(* IEC 61131-3 sources: AutomationLab/ConveyerObject, 5 files *)

(* ---- ConveyerType.st ---- *)
TYPE ConveyerType :
STRUCT
	SensorA : BOOL;
	ComRotateLent : BOOL;
END_STRUCT
END_TYPE

(* ---- DT_Conveyer.st ---- *)
TYPE DT_Conveyer:
STRUCT
	// Коробка на конце ленты (от оптического датчика)
	BoxOnEndPosition: BOOL;
	// Команда на вращение ленты
	ComRotateLent: BOOL;
END_STRUCT
END_TYPE

(* ---- Conveyer_Main.st ---- *)
// ============================================
// ФУНКЦИОНАЛЬНЫЙ БЛОК — конвейер
// ============================================
FUNCTION_BLOCK Conveyer_Main
VAR_INPUT
END_VAR

VAR_OUTPUT
END_VAR

VAR
    conveyerData: ConveyerType; // данные конвейера
    conveyer: Conveyer1; // блок управления конвейером
    hard: G_Hardware; // обмен с аппаратурой
    inter: G_Interface; // сопряжение с лампой оператора
END_VAR

BEGIN
    // обмен с аппаратурой — чтение GVL → ConveyerData, ConveyerData → запись в GVL
    hard(
        ConveyerData := conveyerData
    );

    // вызов блока управления конвейером
    conveyer(
        SensorA := conveyerData.SensorA,
        RotateLent => conveyerData.ComRotateLent
    );

    // сопряжение с лампой оператора — ConveyerData → GVL HMI
    inter(
        ConveyerData := conveyerData
    );

END_FUNCTION_BLOCK

(* ---- Main.st ---- *)
FUNCTION_BLOCK Main
VAR_INPUT
END_VAR
VAR_OUTPUT
END_VAR
VAR
    // Данные конвейера (каталог объекта)
    data: ConveyerType;
    // Алгоритмический блок обработки конвейера
    conveyer: Conveyer;
    // Блок сопряжения с аппаратурой
    hard: Hardware;
END_VAR

// ============================================
// Технологический объект конвейер
// ============================================

// Циклическое выполнение алгоритма
conveyer(Data := data);

// Подключение блока хардвар
hard(SensorA:= GVL.DI_SensorA, ComMotor=> GVL.DO_ComMotor, Data:= data);

(* ---- MainConveyer_FB.st ---- *)
FUNCTION_BLOCK MainConveyer_FB
VAR_INPUT
END_VAR
VAR_OUTPUT
END_VAR
VAR
    // Данные конвейера (каталог объекта)
    data: ConveyerType;
    // Алгоритмический блок обработки конвейера
    conveyer: Conveyer_FB;
END_VAR

// Циклическое выполнение алгоритма
conveyer(Data := data);
